(* IEC 61131-3 sources: volt/packages/volt-lsp-iec/test-corpus/lenze-mid/Device/Plc Logic/Application/Library Manager/IODrvEtherCAT, 86 files *)

(* ---- CAA_FILENAME.dut ---- *)
TYPE CAA_FILENAME : CAA.FILENAME;
END_TYPE

(* ---- CAA_PVOID.dut ---- *)
TYPE CAA_PVOID : CAA.PVOID;
END_TYPE

(* ---- CAA_SIZE.dut ---- *)
TYPE CAA_SIZE : CAA.SIZE;
END_TYPE

(* ---- L_ETC_CLEARCOUNTER_COUNTER.dut ---- *)
TYPE L_ETC_CLEARCOUNTER_COUNTER :
(
	NONE := 0,
	COUNTER_MASTER := 1,
	COUNTER_SLAVE := 2,
	COUNTER_ALL := 3
);
END_TYPE

(* ---- L_ETC_CMD_T.dut ---- *)
TYPE L_ETC_CMD_T :
STRUCT
	CMD : UDINT;
	RESULT : UDINT;
END_STRUCT
END_TYPE

(* ---- L_ETC_COE_EMERGENCY.dut ---- *)
TYPE L_ETC_COE_EMERGENCY :
STRUCT
	UIDEVICE : UINT;
	DTTIMESTAMP : DATE_AND_TIME;
	WERRORCODE : WORD;
	BYERRORREGISTER : BYTE;
	ABYDATA : ARRAY [0..4] OF BYTE;
END_STRUCT
END_TYPE

(* ---- L_ETC_COE_EMERGENCY_BUFFER_DATA.dut ---- *)
TYPE L_ETC_COE_EMERGENCY_BUFFER_DATA :
STRUCT
	STRUCTEMERGENCY : L_ETC_COE_EMERGENCY;
	BBUFFEROVERFLOW : BOOL;
END_STRUCT
END_TYPE

(* ---- L_ETC_COE_FLAGS.dut ---- *)
TYPE L_ETC_COE_FLAGS :
(
	ETC_E_COMPLETEACCESS := 16#1
);
END_TYPE

(* ---- L_ETC_DIAGNOSTIC.dut ---- *)
TYPE L_ETC_DIAGNOSTIC :
STRUCT
	WSTATE : L_ETC_STATE;
	STSTATE : STRING;
	XETHERNETLINKUP : BOOL;
	XNOTALLSLAVESOPERATIONAL : BOOL;
	UDIFRAMECOUNTER : UDINT;
	UDIFRAMERESPONSEERRORCOUNTER : UDINT;
	UDICYCWORKINGCOUNTERERRORCOUNTER : UDINT;
	XBUSMISMATCH : BOOL;
	UINUMBEROFSLAVESFOUND : UINT;
	UINUMBEROFSLAVESCONFIGURED : UINT;
	DWLASTERRORCODE : DWORD;
	STLASTERROR : STRING;
	XDC_ENABLED : BOOL;
	XDC_INSYNC : BOOL;
	XDC_BUSY : BOOL;
	DIDC_CURRENTDEVIATION : DINT;
	UDIEMERGENCYNO : UDINT;
END_STRUCT
END_TYPE

(* ---- L_ETC_ENGMODE_STATE.dut ---- *)
TYPE L_ETC_ENGMODE_STATE :
(
	NORMAL := 0,
	ENTERENGMODE := 1,
	ENGMODE := 2,
	LEAVINGENGMODE := 3
);
END_TYPE

(* ---- L_ETC_ERRORCODE.dut ---- *)
TYPE L_ETC_ERRORCODE :
(
	ETC_E_NOERROR := 16#0,
	ETC_E_ERROR := 16#98110000,
	ETC_EMRAS_E_ERROR := 16#98110180,
	ETC_DCM_E_ERROR := 16#981201C0,
	ETC_TEXTBASE := 16#200,
	ETC_ALSTATEBASE := 16#300,
	ETC_E_NOTSUPPORTED := 16#98110001,
	ETC_E_INVALIDINDEX := 16#98110002,
	ETC_E_INVALIDOFFSET := 16#98110003,
	ETC_E_INVALIDSIZE := 16#98110005,
	ETC_E_INVALIDDATA := 16#98110006,
	ETC_E_NOTREADY := 16#98110007,
	ETC_E_BUSY := 16#98110008,
	ETC_E_ACYC_FRM_FREEQ_EMPTY := 16#98110009,
	ETC_E_NOMEMORY := 16#9811000A,
	ETC_E_INVALIDPARM := 16#9811000B,
	ETC_E_NOTFOUND := 16#9811000C,
	ETC_E_INVALIDSTATE := 16#9811000E,
	ETC_E_TIMER_LIST_FULL := 16#9811000F,
	ETC_E_TIMEOUT := 16#98110010,
	ETC_E_OPENFAILED := 16#98110011,
	ETC_E_SENDFAILED := 16#98110012,
	ETC_E_INSERTMAILBOX := 16#98110013,
	ETC_E_INVALIDCMD := 16#98110014,
	ETC_E_UNKNOWN_MBX_PROTOCOL := 16#98110015,
	ETC_E_ACCESSDENIED := 16#98110016,
	ETC_E_PRODKEY_INVALID := 16#9811001A,
	ETC_E_WRONG_FORMAT := 16#9811001B,
	ETC_E_FEATURE_DISABLED := 16#9811001C,
	ETC_E_SHADOW_MEMORY := 16#9811001D,
	ETC_E_BUSCONFIG_MISMATCH := 16#9811001E,
	ETC_E_CONFIGDATAREAD := 16#9811001F,
	ETC_E_XML_CYCCMDS_MISSING := 16#98110021,
	ETC_E_XML_ALSTATUS_READ_MISSING := 16#98110022,
	ETC_E_MCSM_FATAL_ERROR := 16#98110023,
	ETC_E_SLAVE_ERROR := 16#98110024,
	ETC_E_FRAME_LOST := 16#98110025,
	ETC_E_CMD_MISSING := 16#98110026,
	ETC_E_INVALID_DCL_MODE := 16#98110028,
	ETC_E_AI_ADDRESS := 16#98110029,
	ETC_E_INVALID_SLAVE_STATE := 16#9811002A,
	ETC_E_SLAVE_NOT_ADDRESSABLE := 16#9811002B,
	ETC_E_CYC_CMDS_OVERFLOW := 16#9811002C,
	ETC_E_LINK_DISCONNECTED := 16#9811002D,
	ETC_E_MASTERCORE_INACCESSIBLE := 16#9811002E,
	ETC_E_COE_MBXSND_WKC_ERROR := 16#9811002F,
	ETC_E_COE_MBXRCV_WKC_ERROR := 16#98110030,
	ETC_E_NO_MBX_SUPPORT := 16#98110031,
	ETC_E_NO_COE_SUPPORT := 16#98110032,
	ETC_E_NO_EOE_SUPPORT := 16#98110033,
	ETC_E_NO_FOE_SUPPORT := 16#98110034,
	ETC_E_NO_SOE_SUPPORT := 16#98110035,
	ETC_E_NO_VOE_SUPPORT := 16#98110036,
	ETC_E_EVAL_VIOLATION := 16#98110037,
	ETC_E_EVAL_EXPIRED := 16#98110038,
	ETC_E_SDO_ABORTCODE_TOGGLE := 16#98110040,
	ETC_E_SDO_ABORTCODE_TIMEOUT := 16#98110041,
	ETC_E_SDO_ABORTCODE_CCS_SCS := 16#98110042,
	ETC_E_SDO_ABORTCODE_BLK_SIZE := 16#98110043,
	ETC_E_SDO_ABORTCODE_SEQNO := 16#98110044,
	ETC_E_SDO_ABORTCODE_CRC := 16#98110045,
	ETC_E_SDO_ABORTCODE_MEMORY := 16#98110046,
	ETC_E_SDO_ABORTCODE_ACCESS := 16#98110047,
	ETC_E_SDO_ABORTCODE_WRITEONLY := 16#98110048,
	ETC_E_SDO_ABORTCODE_READONLY := 16#98110049,
	ETC_E_SDO_ABORTCODE_INDEX := 16#9811004A,
	ETC_E_SDO_ABORTCODE_PDO_MAP := 16#9811004B,
	ETC_E_SDO_ABORTCODE_PDO_LEN := 16#9811004C,
	ETC_E_SDO_ABORTCODE_P_INCOMP := 16#9811004D,
	ETC_E_SDO_ABORTCODE_I_INCOMP := 16#9811004E,
	ETC_E_SDO_ABORTCODE_HARDWARE := 16#9811004F,
	ETC_E_SDO_ABORTCODE_DATA_SIZE := 16#98110050,
	ETC_E_SDO_ABORTCODE_DATA_SIZE1 := 16#98110051,
	ETC_E_SDO_ABORTCODE_DATA_SIZE2 := 16#98110052,
	ETC_E_SDO_ABORTCODE_OFFSET := 16#98110053,
	ETC_E_SDO_ABORTCODE_DATA_RANGE := 16#98110054,
	ETC_E_SDO_ABORTCODE_DATA_RANGE1 := 16#98110055,
	ETC_E_SDO_ABORTCODE_DATA_RANGE2 := 16#98110056,
	ETC_E_SDO_ABORTCODE_MINMAX := 16#98110057,
	ETC_E_SDO_ABORTCODE_GENERAL := 16#98110058,
	ETC_E_SDO_ABORTCODE_TRANSFER := 16#98110059,
	ETC_E_SDO_ABORTCODE_TRANSFER1 := 16#9811005A,
	ETC_E_SDO_ABORTCODE_TRANSFER2 := 16#9811005B,
	ETC_E_SDO_ABORTCODE_DICTIONARY := 16#9811005C,
	ETC_E_SDO_ABORTCODE_UNKNOWN := 16#9811005D,
	ETC_E_FOE_ERRCODE_NOTDEFINED := 16#98110060,
	ETC_E_FOE_ERRCODE_NOTFOUND := 16#98110061,
	ETC_E_FOE_ERRCODE_ACCESS := 16#98110062,
	ETC_E_FOE_ERRCODE_DISKFULL := 16#98110063,
	ETC_E_FOE_ERRCODE_ILLEGAL := 16#98110064,
	ETC_E_FOE_ERRCODE_PACKENO := 16#98110065,
	ETC_E_FOE_ERRCODE_EXISTS := 16#98110066,
	ETC_E_FOE_ERRCODE_NOUSER := 16#98110067,
	ETC_E_FOE_ERRCODE_BOOTSTRAPONLY := 16#98110068,
	ETC_E_FOE_ERRCODE_NOTINBOOTSTRAP := 16#98110069,
	ETC_E_FOE_ERRCODE_INVALIDPASSWORD := 16#9811006A,
	ETC_E_FOE_ERRCODE_PROGERROR := 16#9811006B,
	ETC_E_CFGFILENOTFOUND := 16#98110070,
	ETC_E_EEPROMREADERROR := 16#98110071,
	ETC_E_EEPROMWRITEERROR := 16#98110072,
	ETC_E_XML_CYCCMDS_SIZEMISMATCH := 16#98110073,
	ETC_E_XML_INVALID_INP_OFF := 16#98110074,
	ETC_E_XML_INVALID_OUT_OFF := 16#98110075,
	ETC_E_PORTCLOSE := 16#98110076,
	ETC_E_PORTOPEN := 16#98110077,
	ETC_E_SOE_ERRORCODE_INVALID_ACCESS := 16#98110078,
	ETC_E_SOE_ERRORCODE_NOT_EXIST := 16#98110079,
	ETC_E_SOE_ERRORCODE_INVL_ACC_ELEM1 := 16#9811007A,
	ETC_E_SOE_ERRORCODE_NAME_NOT_EXIST := 16#9811007B,
	ETC_E_SOE_ERRORCODE_NAME_UNDERSIZE := 16#9811007C,
	ETC_E_SOE_ERRORCODE_NAME_OVERSIZE := 16#9811007D,
	ETC_E_SOE_ERRORCODE_NAME_UNCHANGE := 16#9811007E,
	ETC_E_SOE_ERRORCODE_NAME_WR_PROT := 16#9811007F,
	ETC_E_SOE_ERRORCODE_UNDERS_TRANS := 16#98110080,
	ETC_E_SOE_ERRORCODE_OVERS_TRANS := 16#98110081,
	ETC_E_SOE_ERRORCODE_ATTR_UNCHANGE := 16#98110082,
	ETC_E_SOE_ERRORCODE_ATTR_WR_PROT := 16#98110083,
	ETC_E_SOE_ERRORCODE_UNIT_NOT_EXIST := 16#98110084,
	ETC_E_SOE_ERRORCODE_UNIT_UNDERSIZE := 16#98110085,
	ETC_E_SOE_ERRORCODE_UNIT_OVERSIZE := 16#98110086,
	ETC_E_SOE_ERRORCODE_UNIT_UNCHANGE := 16#98110087,
	ETC_E_SOE_ERRORCODE_UNIT_WR_PROT := 16#98110088,
	ETC_E_SOE_ERRORCODE_MIN_NOT_EXIST := 16#98110089,
	ETC_E_SOE_ERRORCODE_MIN_UNDERSIZE := 16#9811008A,
	ETC_E_SOE_ERRORCODE_MIN_OVERSIZE := 16#9811008B,
	ETC_E_SOE_ERRORCODE_MIN_UNCHANGE := 16#9811008C,
	ETC_E_SOE_ERRORCODE_MIN_WR_PROT := 16#9811008D,
	ETC_E_SOE_ERRORCODE_MAX_NOT_EXIST := 16#9811008E,
	ETC_E_SOE_ERRORCODE_MAX_UNDERSIZE := 16#9811008F,
	ETC_E_SOE_ERRORCODE_MAX_OVERSIZE := 16#98110090,
	ETC_E_SOE_ERRORCODE_MAX_UNCHANGE := 16#98110091,
	ETC_E_SOE_ERRORCODE_MAX_WR_PROT := 16#98110092,
	ETC_E_SOE_ERRORCODE_DATA_NOT_EXIST := 16#98110093,
	ETC_E_SOE_ERRORCODE_DATA_UNDERSIZE := 16#98110094,
	ETC_E_SOE_ERRORCODE_DATA_OVERSIZE := 16#98110095,
	ETC_E_SOE_ERRORCODE_DATA_UNCHANGE := 16#98110096,
	ETC_E_SOE_ERRORCODE_DATA_WR_PROT := 16#98110097,
	ETC_E_SOE_ERRORCODE_DATA_MIN_LIMIT := 16#98110098,
	ETC_E_SOE_ERRORCODE_DATA_MAX_LIMIT := 16#98110099,
	ETC_E_SOE_ERRORCODE_DATA_INCOR := 16#9811009A,
	ETC_E_SOE_ERRORCODE_PASWD_PROT := 16#9811009B,
	ETC_E_SOE_ERRORCODE_TEMP_UNCHANGE := 16#9811009C,
	ETC_E_SOE_ERRORCODE_INVL_INDIRECT := 16#9811009D,
	ETC_E_SOE_ERRORCODE_TEMP_UNCHANGE1 := 16#9811009E,
	ETC_E_SOE_ERRORCODE_ALREADY_ACTIVE := 16#9811009F,
	ETC_E_SOE_ERRORCODE_NOT_INTERRUPT := 16#98110100,
	ETC_E_SOE_ERRORCODE_CMD_NOT_AVAIL := 16#98110101,
	ETC_E_SOE_ERRORCODE_CMD_NOT_AVAIL1 := 16#98110102,
	ETC_E_SOE_ERRORCODE_DRIVE_NO := 16#98110103,
	ETC_E_SOE_ERRORCODE_IDN := 16#98110104,
	ETC_E_SOE_ERRORCODE_FRAGMENT_LOST := 16#98110105,
	ETC_E_SOE_ERRORCODE_BUFFER_FULL := 16#98110106,
	ETC_E_SOE_ERRORCODE_NO_DATA := 16#98110107,
	ETC_E_SOE_ERRORCODE_NO_DEFAULT_VALUE := 16#98110108,
	ETC_E_SOE_ERRORCODE_DEFAULT_LONG := 16#98110109,
	ETC_E_SOE_ERRORCODE_DEFAULT_WP := 16#9811010A,
	ETC_E_SOE_ERRORCODE_INVL_DRIVE_NO := 16#9811010B,
	ETC_E_SOE_ERRORCODE_GENERAL_ERROR := 16#9811010C,
	ETC_E_SOE_ERRCODE_NO_ELEM_ADR := 16#9811010D,
	ETC_E_SLAVE_NOT_PRESENT := 16#9811010E,
	ETC_E_NO_FOE_SUPPORT_BS := 16#9811010F,
	ETC_E_EEPROMRELOADERROR := 16#98110110,
	ETC_E_SLAVECTRLRESETERROR := 16#98110111,
	ETC_E_SYSDRIVERMISSING := 16#98110112,
	ETC_E_BUSCONFIG_TOPOCHANGE := 16#9811011E,
	ETC_E_EOE_MBX_WKC_ERROR := 16#9811011F,
	ETC_E_FOE_MBX_WKC_ERROR := 16#98110120,
	ETC_E_SOE_MBX_WKC_ERROR := 16#98110121,
	ETC_E_AOE_MBX_WKC_ERROR := 16#98110122,
	ETC_E_VOE_MBX_WKC_ERROR := 16#98110123,
	ETC_E_EEPROMASSIGNERROR := 16#98110124,
	ETC_E_MBX_ERROR_TYPE := 16#98110125,
	ETC_DCM_E_NOTINITIALIZED := 16#981201C1,
	ETC_DCM_E_MAX_CTL_ERROR_EXCEED := 16#981201C2,
	ETC_DCM_E_NOMEMORY := 16#981201C3,
	ETC_DCM_E_INVALID_HWLAYER := 16#981201C4,
	ETC_DCM_E_TIMER_MODIFY_ERROR := 16#981201C5,
	ETC_DCM_E_TIMER_NOT_RUNNING := 16#981201C6,
	ETC_DCM_E_WRONG_CPU := 16#981201C7,
	ETC_DCM_E_INVALID_SYNC_PERIOD := 16#981201C8,
	ETC_DCM_E_INVALID_SETVAL := 16#981201C9,
	ETC_DCM_E_DRIFT_TO_HIGH := 16#981201CA,
	ETC_EMRAS_E_INVALIDCOOKIE := 16#98110181,
	ETC_EMRAS_E_MULSRVDISMULCON := 16#98110183,
	ETC_EMRAS_E_LOGONCANCELLED := 16#98110184,
	ETC_EMRAS_E_INVALIDVERSION := 16#98110186,
	ETC_EMRAS_E_INVALIDACCESSCONFIG := 16#98110187,
	ETC_EMRAS_E_ACCESSLESS := 16#98110188,
	ETC_EMRAS_EVT_SERVERSTOPPED := 16#98110191,
	ETC_EMRAS_EVT_WDEXPIRED := 16#98110192,
	ETC_EMRAS_EVT_RECONEXPIRED := 16#98110193,
	ETC_EMRAS_EVT_CLIENTLOGON := 16#98110194,
	ETC_EMRAS_EVT_RECONNECT := 16#98110195,
	ETC_EMRAS_EVT_SOCKCHANGE := 16#98110196,
	ETC_EMRAS_EVT_CLNTDISC := 16#98110197
);
END_TYPE

(* ---- L_ETC_EVTPARAM_PARAMETERTRANSFER.dut ---- *)
TYPE L_ETC_EVTPARAM_PARAMETERTRANSFER :
STRUCT
	WSERVICE : WORD;
	UIDEVICE : WORD;
	DWRESULT : DWORD;
END_STRUCT
END_TYPE

(* ---- L_ETC_HC_GROUPSTATESUMMARY.dut ---- *)
TYPE L_ETC_HC_GROUPSTATESUMMARY :
(
	ETC_STATE_NONE := 16#0,
	ETC_STATE_INIT := 16#1,
	ETC_STATE_PREOPERATIONAL := 16#2,
	ETC_STATE_SAVEOPERATIONAL := 16#4,
	ETC_STATE_OPERATIONAL := 16#8,
	ETC_STATE_SLAVE_MISSING := 16#100,
	ETC_STATE_BOOTSTRAP := 16#700
);
END_TYPE

(* ---- L_ETC_HC_ROLE.dut ---- *)
TYPE L_ETC_HC_ROLE :
(
	HC_ROLE_STATIC := 16#0,
	HC_ROLE_HEAD := 16#1,
	HC_ROLE_MEMBER := 16#2
);
END_TYPE

(* ---- L_ETC_IOCTLOPARMS.dut ---- *)
TYPE L_ETC_IOCTLOPARMS :
STRUCT
	PBYINBUF : POINTER TO BYTE;
	DWINBUFSIZE : DWORD;
	PBYOUTBUF : POINTER TO BYTE;
	DWOUTBUFSIZE : DWORD;
	PDWNUMOUTDATA : POINTER TO DWORD;
END_STRUCT
END_TYPE

(* ---- L_ETC_LANGUAGE.dut ---- *)
TYPE L_ETC_LANGUAGE :
(
	ENG,
	DE
);
END_TYPE

(* ---- L_ETC_MMCSERVICE.dut ---- *)
TYPE L_ETC_MMCSERVICE :
(
	NONE := 0,
	RUN_WITHOUT_CHECK := 16#1,
	RUN_OPTIONAL_SLAVES_ALLOWED := 16#2,
	RUN_OPTIONAL_SLAVES_PROHIBITED := 16#3,
	ADDR_ASSIGNMENT_EXTERNALLY := 16#100,
	ADDR_ASSIGNMENT_CONFIG_SLAVEORDER := 16#200,
	ADDR_ASSIGNMENT_CONFIG_PARAMETER := 16#300
);
END_TYPE

(* ---- L_ETC_MMCSERVICEERROR.dut ---- *)
TYPE L_ETC_MMCSERVICEERROR :
(
	NO_ERROR := 16#0,
	CONFIG_INVALID := 16#1,
	CONFIG_FILE_ERROR := 16#2,
	IDENT_FILE_ERROR := 16#3,
	SERVICE_INVALID := 16#100,
	SERVICE_INVALID_STATE := 16#101,
	ADDR_INTERNAL_ERROR := 16#10000,
	ADDR_NO_MEMORY := 16#10001,
	ADDR_LESS_CONNECTED := 16#10002,
	ADDR_MORE_CONNECTED := 16#10003,
	ADDR_UNEXPECTED_DEVICE := 16#10004,
	ADDR_ASSIGN_ERROR := 16#10005,
	ADDR_NO_SLAVES_CONNECTED := 16#10006
);
END_TYPE

(* ---- L_ETC_MMCSERVICESTATE.dut ---- *)
TYPE L_ETC_MMCSERVICESTATE :
(
	STOPPED,
	RUNNING,
	NOT_READY := 16#FFFF
);
END_TYPE

(* ---- L_ETC_PARAMETERTRANSFERSERVICE_CODE.dut ---- *)
TYPE L_ETC_PARAMETERTRANSFERSERVICE_CODE :
(
	START := WORD#16#1,
	STATE := WORD#16#2,
	DONE := WORD#16#4,
	ABORT := WORD#16#8000
);
END_TYPE

(* ---- L_ETC_SLAVE_PORTS.dut ---- *)
TYPE L_ETC_SLAVE_PORTS :
STRUCT
	PORT0 : BYTE;
	PORT1 : BYTE;
	PORT2 : BYTE;
	PORT3 : BYTE;
END_STRUCT
END_TYPE

(* ---- L_ETC_SLAVE_PORTS2.dut ---- *)
TYPE L_ETC_SLAVE_PORTS2 :
STRUCT
	PORT0 : WORD;
	PORT1 : WORD;
	PORT2 : WORD;
	PORT3 : WORD;
END_STRUCT
END_TYPE

(* ---- L_ETC_SLVSTATISTICS_DESC2_T.dut ---- *)
TYPE L_ETC_SLVSTATISTICS_DESC2_T :
STRUCT
	ABYINVALIDFRAMECNT : ARRAY [0..3] OF BYTE;
	ABYRXERRORCNT : ARRAY [0..3] OF BYTE;
	ABYFWDRXERRORCNT : ARRAY [0..3] OF BYTE;
	BYPROCESSINGUNITERRORCNT : BYTE;
	BYPDIERRORCNT : BYTE;
	WALSTATUSCODE : WORD;
	ABYLOSTLINKCNT : ARRAY [0..3] OF BYTE;
	QWREADTIME : ULINT;
	QWCHANGETIME : ULINT;
END_STRUCT
END_TYPE

(* ---- L_ETC_SLVSTATISTICS_DESC_T.dut ---- *)
TYPE L_ETC_SLVSTATISTICS_DESC_T :
STRUCT
	ABYINVALIDFRAMECNT : ARRAY [0..3] OF BYTE;
	ABYRXERRORCNT : ARRAY [0..3] OF BYTE;
	ABYFWDRXERRORCNT : ARRAY [0..3] OF BYTE;
	BYPROCESSINGUNITERRORCNT : BYTE;
	BYPDIERRORCNT : BYTE;
	WALSTATUSCODE : WORD;
	ABYLOSTLINKCNT : ARRAY [0..3] OF BYTE;
END_STRUCT
END_TYPE

(* ---- L_ETC_STATE.dut ---- *)
TYPE L_ETC_STATE :
(
	ETC_STATE_NONE := 16#0,
	ETC_STATE_INIT := 16#1,
	ETC_STATE_PREOPERATIONAL := 16#2,
	ETC_STATE_BOOT := 16#3,
	ETC_STATE_SAVEOPERATIONAL := 16#4,
	ETC_STATE_OPERATIONAL := 16#8,
	ETC_STATE_UNKNOWN := 16#FFEF
);
END_TYPE

(* ---- ETC_CONSTANTS.gvl ---- *)
VAR_GLOBAL
	_ETC_NUMBER_OF_MASTERS : INT := 1;
	_ETC_NUMBER_OF_SLAVES : INT := 9;
	_ETC_NUMBER_OF_SDO : INT := 676;
	_ETC_NUMBER_OF_INPUT_BYTES : INT := 511;
	_ETC_NUMBER_OF_OUTPUT_BYTES : INT := 511;
	_ETC_SYSTEM_HAS_INTEL_BYTEORDER : BOOL := TRUE;
END_VAR

(* ---- L_ETC_GLOBALS.gvl ---- *)
VAR_GLOBAL
	L_ETC_CMPID_IODRVETC : UDINT := 16#2006;
	L_ETC_EVT_PARAMETERTRANSFER_SERVICE : UDINT := 16#10000003;
END_VAR

(* ---- L_ETC_HC_GROUP_ITF.itf ---- *)
INTERFACE L_ETC_HC_GROUP_ITF
END_INTERFACE

(* ---- GETBOOLEANPROPERTY.pou ---- *)
FUNCTION GETBOOLEANPROPERTY : BOOL
VAR_INPUT
	STKEY : WSTRING;
END_VAR
END_FUNCTION

(* ---- GETCOMPANY.pou ---- *)
FUNCTION GETCOMPANY : WSTRING
END_FUNCTION

(* ---- GETNUMBERPROPERTY.pou ---- *)
FUNCTION GETNUMBERPROPERTY : DINT
VAR_INPUT
	STKEY : WSTRING;
END_VAR
END_FUNCTION

(* ---- GETTEXTPROPERTY.pou ---- *)
FUNCTION GETTEXTPROPERTY : WSTRING
VAR_INPUT
	STKEY : WSTRING;
END_VAR
END_FUNCTION

(* ---- GETTEXTPROPERTY2.pou ---- *)
FUNCTION GETTEXTPROPERTY2 : POINTER TO WSTRING
VAR_INPUT
	STKEY : WSTRING;
END_VAR
END_FUNCTION

(* ---- GETTITLE.pou ---- *)
FUNCTION GETTITLE : WSTRING
END_FUNCTION

(* ---- GETVERSION.pou ---- *)
FUNCTION GETVERSION : VERSION
END_FUNCTION

(* ---- GETVERSIONPROPERTY.pou ---- *)
FUNCTION GETVERSIONPROPERTY : VERSION
VAR_INPUT
	STKEY : WSTRING;
END_VAR
END_FUNCTION

(* ---- L_ETC_GETERRORSTRING.pou ---- *)
FUNCTION L_ETC_GETERRORSTRING : STRING(256)
VAR_INPUT
	EERRORCODE : L_ETC_ERRORCODE;
	ELANGUAGE : L_ETC_LANGUAGE := eng;
END_VAR
END_FUNCTION

(* ---- L_ETC_GETMASTER.pou ---- *)
FUNCTION L_ETC_GETMASTER : POINTER TO L_IODrvEtherCAT
VAR_INPUT
	USICOM : USINT;
END_VAR
END_FUNCTION

(* ---- L_ETC_GETSLAVE.pou ---- *)
FUNCTION L_ETC_GETSLAVE : POINTER TO ETCSlave
VAR_INPUT
	UIDEVICE : UINT;
END_VAR
END_FUNCTION

(* ---- L_ETC_HC_GETGROUP.pou ---- *)
FUNCTION L_ETC_HC_GETGROUP : L_ETC_HC_GROUP_ITF
VAR_INPUT
	USICOM : USINT := 1;
	GROUPNUMBER : UINT;
END_VAR
END_FUNCTION

(* ---- L_ETC_HC_GETGROUPCOUNT.pou ---- *)
FUNCTION L_ETC_HC_GETGROUPCOUNT : UINT
VAR_INPUT
	USICOM : USINT := 1;
END_VAR
END_FUNCTION

(* ---- L_ETC_HC_GETSLAVESOFGROUP.pou ---- *)
FUNCTION L_ETC_HC_GETSLAVESOFGROUP : DWORD
VAR_INPUT
	USICOM : USINT := 1;
	GROUPNUMBER : UINT;
	COUNT : POINTER TO UINT;
	SLAVES : POINTER TO POINTER TO ETCSlave;
END_VAR
END_FUNCTION

(* ---- L_ETC_IOCONTROL.pou ---- *)
FUNCTION L_ETC_IOCONTROL : DWORD
VAR_INPUT
	DWCODE : DWORD;
	PPARMS : POINTER TO L_ETC_IOCTLOPARMS;
END_VAR
END_FUNCTION

(* ---- ETCSLAVE.pou ---- *)
FUNCTION_BLOCK ETCSLAVE
VAR_INPUT
	XSETOPERATIONAL : BOOL;
END_VAR
VAR_OUTPUT
	XDONE : BOOL;
	XBUSY : BOOL;
	XERROR : BOOL;
	EERRORCODE : L_ETC_ERRORCODE;
	WSTATE : WORD;
END_VAR
VAR
	M_PIOCONFIGCONNECTOR : POINTER TO IoConfigConnector;
	M_SZPATH : STRING;
	M_SZNAME : STRING;
	M_DWVENDORID : DWORD;
	M_DWPRODUCTID : DWORD;
	M_DWREVISIONID : DWORD;
	M_UIPHYSSLAVEADDR : UINT;
	M_XDCENABLE : BOOL;
	M_XSETOPERATIONALLAST : BOOL;
	M_WSLAVESTATEACT : WORD;
	FBSLAVE2 : ETCSlave2;
	M_HCINIT : BOOL;
	M_HCINTERFACE : L_ETC_HC_GROUP_ITF;
	M_HCROLE : L_ETC_HC_ROLE;
	M_PMSSELECTIONPAR : POINTER TO IoStandard.IoConfigParameter;
	M_PMSSELECTION : USINT;
	MODULEHANDLERBASE : L_IMHP_ModuleHandler;
	M_SCOMMPATH : STRING(199);
	SLAVEADDRESS : UINT;
	REGISTERONCOMPONENTDIRECTORY : L_IC1P_RegisterOnComponentDirectory;
	M_ITFEVENTCALLBACK : CmpEventMgr.ICmpEventCallback;
	M_HEVENTUPDATECONFIGURATIONDONE : RTS_IEC_HANDLE;
	M_HINTERFACEUPDATECONFIGURATIONDONE : RTS_IEC_HANDLE;
	DCENABLE : BOOL;
	HCGROUP : L_ETC_HC_GROUP_ITF;
	HCROLE : L_ETC_HC_ROLE;
	IODRVETHERCAT : POINTER TO L_IODrvEtherCAT;
	ISMANDATORY : BOOL;
	ISPRESENT : BOOL;
	MODULEHANDLER : L_IMHP_IModuleHandler;
	NAME : STRING;
	PARAMETERSET : USINT;
	PHYSSLAVEADDR : UINT;
	WCSTATE : BOOL;
END_VAR
END_FUNCTION_BLOCK

METHOD EVENTCALLBACK : UDINT
VAR_INPUT
	PEVENTPARAM : POINTER TO EventParam;
END_VAR
END_METHOD

METHOD FB_EXIT : BOOL
VAR_INPUT
	BINCOPYCODE : BOOL;
END_VAR
END_METHOD

METHOD INITIALIZE : UDINT
VAR_INPUT
	WMODULETYPE : UINT;
	DWINSTANCE : UDINT;
	PCONNECTOR : POINTER TO IoConfigConnector;
END_VAR
END_METHOD

METHOD FB_INIT : BOOL
VAR_INPUT
	BINITRETAINS : BOOL;
	BINCOPYCODE : BOOL;
END_VAR
END_METHOD

(* ---- ETCSLAVE2.pou ---- *)
FUNCTION_BLOCK ETCSLAVE2
VAR_INPUT
	XSETOPERATIONAL : BOOL;
END_VAR
VAR_OUTPUT
	XDONE : BOOL;
	XBUSY : BOOL;
	XERROR : BOOL;
	EERRORCODE : L_ETC_ERRORCODE;
	WSTATE : WORD;
END_VAR
VAR
	M_PIOCONFIGCONNECTOR : POINTER TO IoConfigConnector;
	M_XSETOPERATIONALLAST : BOOL;
	M_UIPHYSSLAVEADDR : UINT;
	M_ADWJOBDATA : ARRAY [0..31] OF DWORD;
	GETSTATE : WORD;
	HCGROUP : L_ETC_HC_GROUP_ITF;
	HCROLE : L_ETC_HC_ROLE;
	IODRVETHERCAT : POINTER TO L_IODrvEtherCAT;
	ISMANDATORY : BOOL;
	PHYSSLAVEADDR : UINT;
END_VAR
END_FUNCTION_BLOCK

METHOD INITIALIZE : UDINT
VAR_INPUT
	WMODULETYPE : UINT;
	DWINSTANCE : UDINT;
	PCONNECTOR : POINTER TO IoConfigConnector;
END_VAR
END_METHOD

METHOD SETETCSLAVE
VAR_INPUT
	PCONNECTOR : POINTER TO IoConfigConnector;
	PETCSLAVE : POINTER TO ETCSlave;
END_VAR
END_METHOD

(* ---- ETCSLAVE_DIAG.pou ---- *)
FUNCTION_BLOCK ETCSLAVE_DIAG EXTENDS ETCSlave
VAR
	M_TREE : CAADiagTreeBase;
	CHILDNODECOUNT : CAA.COUNT;
	CONNECTOR : POINTER TO IoStandard.IoConfigConnector;
	ENABLE : BOOL;
	FIRSTCHILDNODE : DED.INode;
	INDEX : UDINT;
	ISROOTNODE : BOOL;
	NEXTSIBLINGNODE : DED.INode;
	PARENTNODE : DED.INode;
	SIBLINGNODECOUNT : CAA.COUNT;
END_VAR
END_FUNCTION_BLOCK

METHOD GETCHILD : DED.INode
VAR_INPUT
	UDIINDEX : UDINT;
END_VAR
END_METHOD

METHOD GETDEVICEDIAGNOSISINFO : DED.ERROR
VAR_INPUT
	PDATA : CAA.PVOID;
	SZSIZE : CAA.SIZE;
END_VAR
VAR_OUTPUT
	SZCOUNT : CAA.SIZE;
END_VAR
END_METHOD

METHOD GETDEVICEERRORASYNC : DED.PROC_STATE
VAR_INPUT
	ECMD : DED.PROC_CMD;
END_VAR
VAR_OUTPUT
	EERROR : DED.ERROR;
END_VAR
VAR_IN_OUT
	ERIDEVICEERROR : DED.ERROR_INFO;
END_VAR
END_METHOD

METHOD GETDEVICEINFO : DED.ERROR
VAR_IN_OUT
	DEIINFO : DED.DEVICE_INFO;
END_VAR
END_METHOD

METHOD GETDEVICESTATE : DED.DEVICE_STATE
VAR_OUTPUT
	XDIAGNOSISINFOAVAILABLE : BOOL;
	EERROR : DED.ERROR;
END_VAR
END_METHOD

METHOD GETSPECIFICDEVICEERRORASYNC : DED.PROC_STATE
VAR_INPUT
	ECMD : DED.PROC_CMD;
	PDATA : CAA.PVOID;
	SZSIZE : CAA.SIZE;
END_VAR
VAR_OUTPUT
	SZCOUNT : CAA.SIZE;
	EERROR : DED.ERROR;
END_VAR
END_METHOD

METHOD GETSPECIFICDEVICESTATE : DED.ERROR
VAR_INPUT
	PDATA : CAA.PVOID;
	SZSIZE : CAA.SIZE;
END_VAR
VAR_OUTPUT
	SZCOUNT : CAA.SIZE;
END_VAR
END_METHOD

METHOD INITIALIZE_DIAG : UDINT
VAR_INPUT
	PCONNECTOR : POINTER TO IoStandard.IoConfigConnector;
	NCONNECTORCOUNT : DINT;
	PARENT : POINTER TO DED.INode;
	CHILDREN : POINTER TO DED.INode;
	UDICHILDCOUNT : UDINT;
END_VAR
END_METHOD

METHOD SETCOMMUNICATIONSTATE : DED.ERROR
VAR_INPUT
	EREQUESTEDSTATE : DED.DEVICE_TRANSITION_STATE;
END_VAR
END_METHOD

(* ---- GLOBALTEXTLIST.pou ---- *)
FUNCTION_BLOCK GLOBALTEXTLIST
VAR
	M_TEXTLISTFILE : STRING(255);
	_STNAMESPACE : STRING;
END_VAR
END_FUNCTION_BLOCK

(* ---- L_ETC_CLEARCOUNTER.pou ---- *)
FUNCTION_BLOCK L_ETC_CLEARCOUNTER
VAR_INPUT
	XEXECUTE : BOOL;
	ECOUNTER : L_ETC_CLEARCOUNTER_COUNTER;
END_VAR
VAR_OUTPUT
	XDONE : BOOL;
	XBUSY : BOOL;
	XERROR : BOOL;
	EERRORCODE : L_ETC_ERRORCODE;
END_VAR
VAR
	XEXECUTELAST : BOOL;
	ADWJOBDATA : ARRAY [0..31] OF DWORD;
END_VAR
END_FUNCTION_BLOCK

(* ---- L_ETC_COE_SDOREAD.pou ---- *)
FUNCTION_BLOCK L_ETC_COE_SDOREAD
VAR_INPUT
	XEXECUTE : BOOL;
	XABORT : BOOL := FALSE;
	USICOM : USINT := 1;
	UIDEVICE : UINT;
	WINDEX : WORD;
	BYSUBINDEX : BYTE;
	UDITIMEOUT : UDINT;
	PBUFFER : CAA_PVOID := 0;
	SZSIZE : CAA_SIZE := 0;
END_VAR
VAR_OUTPUT
	XDONE : BOOL;
	XBUSY : BOOL;
	XERROR : BOOL;
	EERRORCODE : L_ETC_ERRORCODE;
	UDISDOABORT : UDINT;
	SZDATAREAD : CAA_SIZE;
END_VAR
VAR
	XEXECUTELAST : BOOL;
	ADWJOBDATA : ARRAY [0..31] OF DWORD;
END_VAR
END_FUNCTION_BLOCK

(* ---- L_ETC_COE_SDOREAD4.pou ---- *)
FUNCTION_BLOCK L_ETC_COE_SDOREAD4
VAR_INPUT
	XEXECUTE : BOOL;
	XABORT : BOOL := FALSE;
	USICOM : USINT := 1;
	UIDEVICE : UINT;
	WINDEX : WORD;
	BYSUBINDEX : BYTE;
	UDITIMEOUT : UDINT;
END_VAR
VAR_OUTPUT
	XDONE : BOOL;
	XBUSY : BOOL;
	XERROR : BOOL;
	EERRORCODE : L_ETC_ERRORCODE;
	UDISDOABORT : UDINT;
	ABYDATA : ARRAY [0..3] OF BYTE;
	SZDATAREAD : CAA_SIZE;
END_VAR
VAR
	SDOREAD : L_ETC_CoE_SdoRead;
END_VAR
END_FUNCTION_BLOCK

(* ---- L_ETC_COE_SDOREADEX.pou ---- *)
FUNCTION_BLOCK L_ETC_COE_SDOREADEX
VAR_INPUT
	XEXECUTE : BOOL;
	XABORT : BOOL := FALSE;
	USICOM : USINT := 1;
	UIDEVICE : UINT;
	DWFLAGS : DWORD;
	WINDEX : WORD;
	BYSUBINDEX : BYTE;
	UDITIMEOUT : UDINT;
	PBUFFER : CAA_PVOID := 0;
	SZSIZE : CAA_SIZE := 0;
END_VAR
VAR_OUTPUT
	XDONE : BOOL;
	XBUSY : BOOL;
	XERROR : BOOL;
	EERRORCODE : L_ETC_ERRORCODE;
	UDISDOABORT : UDINT;
	SZDATAREAD : CAA_SIZE;
END_VAR
VAR
	XEXECUTELAST : BOOL;
	ADWJOBDATA : ARRAY [0..31] OF DWORD;
END_VAR
END_FUNCTION_BLOCK

(* ---- L_ETC_COE_SDOWRITE.pou ---- *)
FUNCTION_BLOCK L_ETC_COE_SDOWRITE
VAR_INPUT
	XEXECUTE : BOOL;
	XABORT : BOOL := FALSE;
	USICOM : USINT := 1;
	UIDEVICE : UINT;
	WINDEX : WORD;
	BYSUBINDEX : BYTE;
	UDITIMEOUT : UDINT;
	PBUFFER : CAA_PVOID;
	SZSIZE : CAA_SIZE;
END_VAR
VAR_OUTPUT
	XDONE : BOOL;
	XBUSY : BOOL;
	XERROR : BOOL;
	EERRORCODE : L_ETC_ERRORCODE;
	UDISDOABORT : UDINT;
END_VAR
VAR
	XEXECUTELAST : BOOL;
	ADWJOBDATA : ARRAY [0..31] OF DWORD;
END_VAR
END_FUNCTION_BLOCK

(* ---- L_ETC_COE_SDOWRITE4.pou ---- *)
FUNCTION_BLOCK L_ETC_COE_SDOWRITE4
VAR_INPUT
	XEXECUTE : BOOL;
	XABORT : BOOL := FALSE;
	USICOM : USINT := 1;
	UIDEVICE : UINT;
	WINDEX : WORD;
	BYSUBINDEX : BYTE;
	UDITIMEOUT : UDINT;
	ABYDATA : ARRAY [0..3] OF BYTE;
	USIDATALENGTH : USINT;
END_VAR
VAR_OUTPUT
	XDONE : BOOL;
	XBUSY : BOOL;
	XERROR : BOOL;
	EERRORCODE : L_ETC_ERRORCODE;
	UDISDOABORT : UDINT;
END_VAR
VAR
	USILEN : USINT;
	SDOWRITE : L_ETC_CoE_SdoWrite;
END_VAR
END_FUNCTION_BLOCK

(* ---- L_ETC_COE_SDOWRITEEX.pou ---- *)
FUNCTION_BLOCK L_ETC_COE_SDOWRITEEX
VAR_INPUT
	XEXECUTE : BOOL;
	XABORT : BOOL := FALSE;
	USICOM : USINT := 1;
	UIDEVICE : UINT;
	DWFLAGS : DWORD;
	WINDEX : WORD;
	BYSUBINDEX : BYTE;
	UDITIMEOUT : UDINT;
	PBUFFER : CAA_PVOID;
	SZSIZE : CAA_SIZE;
END_VAR
VAR_OUTPUT
	XDONE : BOOL;
	XBUSY : BOOL;
	XERROR : BOOL;
	EERRORCODE : L_ETC_ERRORCODE;
	UDISDOABORT : UDINT;
END_VAR
VAR
	XEXECUTELAST : BOOL;
	ADWJOBDATA : ARRAY [0..31] OF DWORD;
END_VAR
END_FUNCTION_BLOCK

(* ---- L_ETC_ENGINEERINGMODE.pou ---- *)
FUNCTION_BLOCK L_ETC_ENGINEERINGMODE
VAR_INPUT
	USICOM : USINT := 1;
	XENABLE : BOOL;
END_VAR
VAR_OUTPUT
	XBUSY : BOOL;
	XACTIVE : BOOL;
	XERROR : BOOL;
	EERRORCODE : L_ETC_ERRORCODE;
	ESTATE : L_ETC_ENGMODE_STATE;
END_VAR
VAR
	USTEP : UINT := 0;
	XENABLEPRE : BOOL;
	CMD : L_ETC_CMD_T;
	RESULT : DWORD;
	SMSTATE : UDINT;
	FBMASTER : POINTER TO L_IODrvEtherCAT;
END_VAR
END_FUNCTION_BLOCK

(* ---- L_ETC_FOE_READ.pou ---- *)
FUNCTION_BLOCK L_ETC_FOE_READ
VAR_INPUT
	XEXECUTE : BOOL;
	XABORT : BOOL := FALSE;
	USICOM : USINT := 1;
	UIDEVICE : UINT;
	SFILENAME : CAA_FILENAME := '';
	SZFILENAMELEN : CAA_SIZE := 0;
	DWPASSWD : DWORD;
	UDITIMEOUT : UDINT;
	PBUFFER : CAA_PVOID := 0;
	SZSIZE : CAA_SIZE := 0;
END_VAR
VAR_OUTPUT
	XDONE : BOOL;
	XBUSY : BOOL;
	XERROR : BOOL;
	EERRORCODE : L_ETC_ERRORCODE;
	SZDATAREAD : CAA_SIZE;
END_VAR
VAR
	XEXECUTELAST : BOOL;
	ADWJOBDATA : ARRAY [0..31] OF DWORD;
END_VAR
END_FUNCTION_BLOCK

(* ---- L_ETC_FOE_WRITE.pou ---- *)
FUNCTION_BLOCK L_ETC_FOE_WRITE
VAR_INPUT
	XEXECUTE : BOOL;
	XABORT : BOOL := FALSE;
	USICOM : USINT := 1;
	UIDEVICE : UINT;
	SFILENAME : CAA_FILENAME := '';
	SZFILENAMELEN : CAA_SIZE := 0;
	DWPASSWD : DWORD;
	UDITIMEOUT : UDINT;
	PBUFFER : CAA_PVOID := 0;
	SZSIZE : CAA_SIZE := 0;
END_VAR
VAR_OUTPUT
	XDONE : BOOL;
	XBUSY : BOOL;
	XERROR : BOOL;
	EERRORCODE : L_ETC_ERRORCODE;
END_VAR
VAR
	XEXECUTELAST : BOOL;
	ADWJOBDATA : ARRAY [0..31] OF DWORD;
END_VAR
END_FUNCTION_BLOCK

(* ---- L_ETC_GETEMERGENCY.pou ---- *)
FUNCTION_BLOCK L_ETC_GETEMERGENCY
VAR_INPUT
	USICOM : USINT := 1;
	XEXECUTE : BOOL;
	XRESET : BOOL;
END_VAR
VAR_OUTPUT
	XDONE : BOOL;
	XBUSY : BOOL;
	XERROR : BOOL;
	EERRORCODE : L_ETC_ERRORCODE;
	OEMCY : L_ETC_COE_EMERGENCY;
	UICOUNT : UINT;
END_VAR
VAR
	M_XEXECUTELAST : BOOL;
	M_XRESETLAST : BOOL;
END_VAR
END_FUNCTION_BLOCK

METHOD DEINITIALIZE : BOOL
END_METHOD

METHOD FB_INIT : BOOL
VAR_INPUT
	BINITRETAINS : BOOL;
	BINCOPYCODE : BOOL;
END_VAR
END_METHOD

METHOD FB_EXIT : BOOL
VAR_INPUT
	BINCOPYCODE : BOOL;
END_VAR
END_METHOD

METHOD INITIALIZE : BOOL
END_METHOD

(* ---- L_ETC_GETMASTERDIAGNOSTIC.pou ---- *)
FUNCTION_BLOCK L_ETC_GETMASTERDIAGNOSTIC
VAR_INPUT
	XRESET : BOOL;
END_VAR
VAR_OUTPUT
	XDONE : BOOL;
	XBUSY : BOOL;
	XERROR : BOOL;
	EERRORCODE : L_ETC_ERRORCODE;
	ODIAGNOSTIC : L_ETC_DIAGNOSTIC;
END_VAR
VAR
	M_UDILASTMESSAGEID : UDINT;
	M_XRESETLAST : BOOL;
END_VAR
END_FUNCTION_BLOCK

(* ---- L_ETC_GETMASTERSTATE.pou ---- *)
FUNCTION_BLOCK L_ETC_GETMASTERSTATE
VAR_INPUT
	XEXECUTE : BOOL;
	UDITIMEOUT : UDINT;
END_VAR
VAR_OUTPUT
	XDONE : BOOL;
	XBUSY : BOOL;
	XERROR : BOOL;
	EERRORCODE : L_ETC_ERRORCODE;
	WSTATE : WORD;
END_VAR
VAR
	XEXECUTELAST : BOOL;
	ADWJOBDATA : ARRAY [0..31] OF DWORD;
END_VAR
END_FUNCTION_BLOCK

(* ---- L_ETC_GETSLAVESTATE.pou ---- *)
FUNCTION_BLOCK L_ETC_GETSLAVESTATE
VAR_INPUT
	XEXECUTE : BOOL;
	UIDEVICE : UINT;
	UDITIMEOUT : UDINT;
END_VAR
VAR_OUTPUT
	XDONE : BOOL;
	XBUSY : BOOL;
	XERROR : BOOL;
	EERRORCODE : L_ETC_ERRORCODE;
	WSTATE : WORD;
END_VAR
VAR
	XEXECUTELAST : BOOL;
	ADWJOBDATA : ARRAY [0..31] OF DWORD;
END_VAR
END_FUNCTION_BLOCK

METHOD FB_INIT : BOOL
VAR_INPUT
	BINITRETAINS : BOOL;
	BINCOPYCODE : BOOL;
END_VAR
END_METHOD

(* ---- L_ETC_HC_GROUP.pou ---- *)
FUNCTION_BLOCK L_ETC_HC_GROUP
VAR
	M_HDEVMANAGER : RTS_IEC_HANDLE;
	M_HINTERFACE : L_ETC_HC_GROUP_ITF;
	M_USICOM : USINT := 1;
	M_GROUPNUMBER : UINT;
	M_NAME : STRING;
	M_GROUPHEAD : POINTER TO ETCSlave;
	M_IDENTVALUE : UINT;
	M_SLAVECOUNT : UINT;
	M_SLAVES : POINTER TO ETCSlave;
	M_GROUPPRESENT : BOOL;
	M_GROUPSTATESUMMARY : WORD;
	M_WCSTATE : BOOL;
	M_RESERVE : ARRAY [0..15] OF ULINT;
	GETGROUPHEAD : POINTER TO ETCSlave;
	GETGROUPPRESENT : BOOL;
	GETGROUPSTATESUMMARY : L_ETC_HC_GROUPSTATESUMMARY;
	GETIDENTIFICATIONVALUE : UINT;
	GETNAME : STRING;
	GETSLAVECOUNT : UINT;
	GETSLAVES : POINTER TO ETCSlave;
	GROUPHEAD : POINTER TO ETCSlave;
	GROUPNUMBER : UINT;
	GROUPPRESENT : BOOL;
	GROUPSTATESUMMARY : WORD;
	IDENTIFICATIONVALUE : UINT;
	NAME : STRING;
	SLAVECOUNT : UINT;
	SLAVES : POINTER TO ETCSlave;
	WCSTATE : BOOL;
END_VAR
END_FUNCTION_BLOCK

METHOD FB_INIT : BOOL
VAR_INPUT
	BINITRETAINS : BOOL;
	BINCOPYCODE : BOOL;
END_VAR
END_METHOD

METHOD GETGROUPNUMBER : UINT
VAR_INPUT
	HINTERFACE : L_ETC_HC_GROUP_ITF;
END_VAR
END_METHOD

(* ---- L_ETC_HC_SETGROUPSTATE.pou ---- *)
FUNCTION_BLOCK L_ETC_HC_SETGROUPSTATE
VAR_INPUT
	USICOM : USINT := 1;
	XEXECUTE : BOOL;
	UIGROUP : UINT;
	WSTATE : WORD;
	UDITIMEOUT : UDINT;
END_VAR
VAR_OUTPUT
	XDONE : BOOL;
	XBUSY : BOOL;
	XERROR : BOOL;
	EERRORCODE : L_ETC_ERRORCODE;
END_VAR
VAR
	XEXECUTELAST : BOOL;
	ADWJOBDATA : ARRAY [0..31] OF DWORD;
END_VAR
END_FUNCTION_BLOCK

(* ---- L_ETC_HC_SETSLAVEPORTSTATE.pou ---- *)
FUNCTION_BLOCK L_ETC_HC_SETSLAVEPORTSTATE
VAR_INPUT
	USICOM : USINT := 1;
	XEXECUTE : BOOL;
	UIDEVICE : UINT;
	UIPORT : UINT;
	XCLOSE : BOOL;
	XFORCE : BOOL;
	UDITIMEOUT : UDINT;
END_VAR
VAR_OUTPUT
	XDONE : BOOL;
	XBUSY : BOOL;
	XERROR : BOOL;
	EERRORCODE : L_ETC_ERRORCODE;
END_VAR
VAR
	XEXECUTELAST : BOOL;
	ADWJOBDATA : ARRAY [0..16] OF DWORD;
END_VAR
END_FUNCTION_BLOCK

(* ---- L_ETC_MMCASSIGNADDRESS.pou ---- *)
FUNCTION_BLOCK L_ETC_MMCASSIGNADDRESS
VAR_INPUT
	XEXECUTE : BOOL;
	UIPOSITION : UINT;
	UIDEVICE : UINT;
END_VAR
VAR_OUTPUT
	XDONE : BOOL;
	XBUSY : BOOL;
	XERROR : BOOL;
	EERRORCODE : L_ETC_ERRORCODE;
END_VAR
VAR
	FBEEPROMWRITE : L_ETC_WriteEEPROM_intern;
END_VAR
END_FUNCTION_BLOCK

(* ---- L_ETC_MMCCONTROLLER.pou ---- *)
FUNCTION_BLOCK L_ETC_MMCCONTROLLER
VAR_INPUT
	XEXECUTE : BOOL;
	XABORT : BOOL;
	ESERVICE : L_ETC_MMCSERVICE;
	SZCONFIGURATION : STRING;
	XRESETTOPOLOGYCHANGEDCOUNTER : BOOL;
END_VAR
VAR_OUTPUT
	XDONE : BOOL;
	XBUSY : BOOL;
	XERROR : BOOL;
	EERRORCODE : L_ETC_MMCSERVICEERROR;
	XABORTED : BOOL;
	ESERVICESTATE : L_ETC_MMCSERVICESTATE;
	UDITOPOLOGYCHANGEDCOUNTER : UDINT;
END_VAR
VAR
	FBMMC : L_ETC_MMCController_intern;
	ACTUALCONFIGURATION : STRING;
	RUNNINGSERVICE : L_ETC_MMCSERVICE;
END_VAR
END_FUNCTION_BLOCK

METHOD FB_INIT : BOOL
VAR_INPUT
	BINITRETAINS : BOOL;
	BINCOPYCODE : BOOL;
END_VAR
END_METHOD

(* ---- L_ETC_MMCCONTROLLER_INTERN.pou ---- *)
FUNCTION_BLOCK L_ETC_MMCCONTROLLER_INTERN
VAR_INPUT
	XEXECUTE : BOOL;
	XABORT : BOOL;
	ESERVICE : L_ETC_MMCSERVICE;
	SZCONFIGURATION : STRING;
	XRESETTOPOLOGYCHANGEDCOUNTER : BOOL;
END_VAR
VAR_OUTPUT
	XDONE : BOOL;
	XBUSY : BOOL;
	XERROR : BOOL;
	EERRORCODE : L_ETC_MMCSERVICEERROR;
	XABORTED : BOOL;
	ESERVICESTATE : L_ETC_MMCSERVICESTATE;
	UDITOPOLOGYCHANGEDCOUNTER : UDINT;
END_VAR
VAR
	ESERVICEACT : L_ETC_MMCSERVICE;
	SZCONFIGURATIONACT : STRING;
	XEXECUTEPRE : BOOL;
	XABORTPRE : BOOL;
	XRESETTOPOLOGYCHANGEDCOUNTERPRE : BOOL;
	ADATA : ARRAY [0..31] OF DWORD;
END_VAR
END_FUNCTION_BLOCK

METHOD INITIALIZE
END_METHOD

(* ---- L_ETC_MMCCONTROLLERBUS.pou ---- *)
FUNCTION_BLOCK L_ETC_MMCCONTROLLERBUS
VAR_INPUT
	XEXECUTE : BOOL;
	XABORT : BOOL;
	SZCONFIGURATION : STRING;
	ESERVICE : L_ETC_MMCSERVICE;
	XRESETTOPOLOGYCHANGEDCOUNTER : BOOL;
END_VAR
VAR_OUTPUT
	XDONE : BOOL;
	XBUSY : BOOL;
	XERROR : BOOL;
	XABORTED : BOOL;
	EERRORCODE : L_ETC_MMCSERVICEERROR;
	ESERVICESTATE : L_ETC_MMCSERVICESTATE;
	UDITOPOLOGYCHANGEDCOUNTER : UDINT;
END_VAR
VAR
	FBMMC : L_ETC_MMCController;
	POMASTER : POINTER TO L_IODrvEtherCAT;
	STATE : INT;
	XEXECUTELAST : BOOL;
	XABORTLAST : BOOL;
	FBTIMEOUT : TON;
	XREADY : BOOL;
	ACTUALCONFIGURATION : STRING;
	RUNNINGSERVICE : L_ETC_MMCSERVICE;
END_VAR
END_FUNCTION_BLOCK

METHOD RESETOUTPUTS
END_METHOD

METHOD SETOUTPUTS
VAR_INPUT
	EERRORCODE2 : L_ETC_MMCSERVICEERROR;
END_VAR
END_METHOD

(* ---- L_ETC_MMCREADADDRESS.pou ---- *)
FUNCTION_BLOCK L_ETC_MMCREADADDRESS
VAR_INPUT
	XEXECUTE : BOOL;
	UIDEVICE : UINT;
	UDITIMEOUT : UDINT;
END_VAR
VAR_OUTPUT
	XDONE : BOOL;
	XBUSY : BOOL;
	XERROR : BOOL;
	EERRORCODE : L_ETC_ERRORCODE;
	UIDEVICESSA : UINT;
END_VAR
VAR
	FBEEPROMREAD : L_ETC_ReadEEPROM_intern;
END_VAR
END_FUNCTION_BLOCK

(* ---- L_ETC_READEEPROM_INTERN.pou ---- *)
FUNCTION_BLOCK L_ETC_READEEPROM_INTERN
VAR_INPUT
	XEXECUTE : BOOL;
	USICOM : USINT := 1;
	UIDEVICE : UINT;
	BAUTOINCADDR : BOOL := 0;
	UDITIMEOUT : UDINT;
	UIWORDADDRESS : UINT;
	PBUFFER : CAA_PVOID := 0;
	SZSIZE : CAA_SIZE := 0;
END_VAR
VAR_OUTPUT
	XDONE : BOOL;
	XBUSY : BOOL;
	XERROR : BOOL;
	EERRORCODE : L_ETC_ERRORCODE;
	SZDATAREAD : CAA_SIZE;
END_VAR
VAR
	XEXECUTELAST : BOOL;
	ADWJOBDATA : ARRAY [0..31] OF DWORD;
END_VAR
END_FUNCTION_BLOCK

(* ---- L_ETC_READERRCNT.pou ---- *)
FUNCTION_BLOCK L_ETC_READERRCNT
VAR_INPUT
	XEXECUTE : BOOL;
	UIDEVICE : UINT;
END_VAR
VAR_OUTPUT
	XDONE : BOOL;
	XBUSY : BOOL;
	XERROR : BOOL;
	EERRORCODE : L_ETC_ERRORCODE;
	REDERRCNT : L_ETC_SLAVE_PORTS;
	GREENERRCNT : L_ETC_SLAVE_PORTS;
END_VAR
VAR
	WINDEX : WORD;
	XEXCECUTEOLD : BOOL;
	WSTATE : WORD;
	GETSLAVESTATE : L_ETC_GetSlaveState;
	MYEC_T_IOCTLPARMS : L_ETC_IOCTLOPARMS;
	RESULT : DWORD;
	SDOREAD : L_ETC_CoE_SdoRead;
	WMYDATA : WORD;
	DWMYLENGTH : CAA_SIZE := 2;
	BYSUBCODEOFFSET : BYTE;
END_VAR
END_FUNCTION_BLOCK

(* ---- L_ETC_READERRCNT2.pou ---- *)
FUNCTION_BLOCK L_ETC_READERRCNT2
VAR_INPUT
	XEXECUTE : BOOL;
	UIDEVICE : UINT;
END_VAR
VAR_OUTPUT
	XDONE : BOOL;
	XBUSY : BOOL;
	XERROR : BOOL;
	EERRORCODE : L_ETC_ERRORCODE;
	REDERRCNT : L_ETC_SLAVE_PORTS2;
	GREENERRCNT : L_ETC_SLAVE_PORTS;
END_VAR
VAR
	WINDEX : WORD;
	XEXCECUTEOLD : BOOL;
	WSTATE : WORD;
	GETSLAVESTATE : L_ETC_GetSlaveState;
	MYEC_T_IOCTLPARMS : L_ETC_IOCTLOPARMS;
	RESULT : DWORD;
	SDOREAD : L_ETC_CoE_SdoReadEx;
	WMYDATA : WORD;
	DWMYLENGTH : CAA_SIZE := 2;
	BYSUBCODEOFFSET : BYTE;
	EC_SLAVE_BASE_ADDRESS : WORD := 1001;
	EC_IOCTL_FORCE_SLVSTAT_COLLECTION : DWORD := 44;
	EC_SLAVE_CONF_AND_INFO_OBJECT_0X3000 : WORD := 16#3000;
	EC_MOD_BASE_SUBIDX_RX_ERR_CNT_PORT0 : BYTE := 24;
END_VAR
END_FUNCTION_BLOCK

METHOD RESETOUTPUT
END_METHOD

(* ---- L_ETC_READERRCNTREAD.pou ---- *)
FUNCTION_BLOCK L_ETC_READERRCNTREAD
VAR_INPUT
	USICOM : USINT := 1;
	XEXECUTE : BOOL;
	UIDEVICE : UINT;
END_VAR
VAR_OUTPUT
	XDONE : BOOL;
	XBUSY : BOOL;
	XERROR : BOOL;
	EERRORCODE : L_ETC_ERRORCODE;
	RXERRORCNT : L_ETC_SLAVE_PORTS2;
	FWDRXERRORCNT : L_ETC_SLAVE_PORTS;
	PROCESSINGUNITERRORCNT : BYTE;
	PDIERRORCNT : BYTE;
	LOSTLINKCNT : L_ETC_SLAVE_PORTS;
END_VAR
VAR
	XEXCECUTEOLD : BOOL;
	WSTATE : WORD;
	PSLAVE : POINTER TO ETCSlave;
	DWSLAVEID : DWORD;
	SLAVEDESC : L_ETC_SLVSTATISTICS_DESC2_T;
	OIOCTLPARAMS : L_ETC_IOCTLOPARMS;
	RESULT : DWORD;
	DWREAD : DWORD;
	EC_IOCTL_GET_SLVSTATISTICS : DWORD := 45;
END_VAR
END_FUNCTION_BLOCK

METHOD RESETOUTPUT
END_METHOD

(* ---- L_ETC_READERRCNTUPDATE.pou ---- *)
FUNCTION_BLOCK L_ETC_READERRCNTUPDATE
VAR_INPUT
	USICOM : USINT := 1;
	XEXECUTE : BOOL;
END_VAR
VAR_OUTPUT
	XDONE : BOOL;
	XBUSY : BOOL;
	XERROR : BOOL;
	EERRORCODE : L_ETC_ERRORCODE;
END_VAR
VAR
	XEXCECUTEOLD : BOOL;
	WSTATE : WORD;
	PMASTER : POINTER TO L_IODrvEtherCAT;
	UDICYCLETIME : DWORD;
	OIOCTLRPARAMS : L_ETC_IOCTLOPARMS;
	RESULT : DWORD;
	TIMER : TON;
	TVAL : TIME;
	EC_IOCTL_FORCE_SLVSTAT_COLLECTION : DWORD := 44;
END_VAR
END_FUNCTION_BLOCK

METHOD RESETOUTPUTS
END_METHOD

(* ---- L_ETC_REGISTERREAD.pou ---- *)
FUNCTION_BLOCK L_ETC_REGISTERREAD
VAR_INPUT
	XEXECUTE : BOOL;
	XABORT : BOOL := FALSE;
	USICOM : USINT := 1;
	XAUTOINCADDR : BOOL := 0;
	UIDEVICE : UINT;
	WREGISTER : WORD;
	UDITIMEOUT : UDINT;
	PBUFFER : CAA_PVOID := 0;
	SZSIZE : CAA_SIZE := 0;
END_VAR
VAR_OUTPUT
	XDONE : BOOL;
	XBUSY : BOOL;
	XERROR : BOOL;
	EERRORCODE : L_ETC_ERRORCODE;
	SZDATAREAD : CAA_SIZE;
END_VAR
VAR
	XEXECUTELAST : BOOL;
	ADWJOBDATA : ARRAY [0..31] OF DWORD;
END_VAR
END_FUNCTION_BLOCK

(* ---- L_ETC_REGISTERWRITE.pou ---- *)
FUNCTION_BLOCK L_ETC_REGISTERWRITE
VAR_INPUT
	XEXECUTE : BOOL;
	XABORT : BOOL := FALSE;
	USICOM : USINT := 1;
	XAUTOINCADDR : BOOL := 0;
	UIDEVICE : UINT;
	WREGISTER : WORD;
	UDITIMEOUT : UDINT;
	PBUFFER : CAA_PVOID := 0;
	SZSIZE : CAA_SIZE := 0;
END_VAR
VAR_OUTPUT
	XDONE : BOOL;
	XBUSY : BOOL;
	XERROR : BOOL;
	EERRORCODE : L_ETC_ERRORCODE;
END_VAR
VAR
	XEXECUTELAST : BOOL;
	ADWJOBDATA : ARRAY [0..31] OF DWORD;
END_VAR
END_FUNCTION_BLOCK

(* ---- L_ETC_RESETERRCNT.pou ---- *)
FUNCTION_BLOCK L_ETC_RESETERRCNT
VAR_INPUT
	XEXECUTE : BOOL;
END_VAR
VAR_OUTPUT
	XDONE : BOOL;
	XBUSY : BOOL;
	XERROR : BOOL;
	EERRORCODE : L_ETC_ERRORCODE;
END_VAR
VAR
	XEXCECUTEOLD : BOOL := 0;
	WSTATE : WORD;
	GETMASTERSTATE : L_ETC_GetMasterState;
	MYEC_T_IOCTLPARMS : L_ETC_IOCTLOPARMS;
	RESULT : DWORD := 0;
END_VAR
END_FUNCTION_BLOCK

(* ---- L_ETC_SETMASTERSTATE.pou ---- *)
FUNCTION_BLOCK L_ETC_SETMASTERSTATE
VAR_INPUT
	XEXECUTE : BOOL;
	WSTATE : WORD;
	UDITIMEOUT : UDINT;
END_VAR
VAR_OUTPUT
	XDONE : BOOL;
	XBUSY : BOOL;
	XERROR : BOOL;
	EERRORCODE : L_ETC_ERRORCODE;
END_VAR
VAR
	XEXECUTELAST : BOOL;
	ADWJOBDATA : ARRAY [0..31] OF DWORD;
END_VAR
END_FUNCTION_BLOCK

(* ---- L_ETC_SETSLAVESTATE.pou ---- *)
FUNCTION_BLOCK L_ETC_SETSLAVESTATE
VAR_INPUT
	XEXECUTE : BOOL;
	UIDEVICE : UINT;
	WSTATE : WORD;
	UDITIMEOUT : UDINT;
END_VAR
VAR_OUTPUT
	XDONE : BOOL;
	XBUSY : BOOL;
	XERROR : BOOL;
	EERRORCODE : L_ETC_ERRORCODE;
END_VAR
VAR
	XEXECUTELAST : BOOL;
	ADWJOBDATA : ARRAY [0..31] OF DWORD;
END_VAR
END_FUNCTION_BLOCK

(* ---- L_ETC_SETSLAVESTATEFWDL.pou ---- *)
FUNCTION_BLOCK L_ETC_SETSLAVESTATEFWDL
VAR_INPUT
	XEXECUTE : BOOL;
	UIDEVICE : UINT;
	WSTATE : WORD;
	UDITIMEOUT : UDINT;
END_VAR
VAR_OUTPUT
	XDONE : BOOL;
	XBUSY : BOOL;
	XERROR : BOOL;
	EERRORCODE : L_ETC_ERRORCODE;
END_VAR
VAR
	XEXECUTELAST : BOOL;
	ADWJOBDATA : ARRAY [0..31] OF DWORD;
END_VAR
END_FUNCTION_BLOCK

(* ---- L_ETC_VOE_WRITEREAD_INTERN.pou ---- *)
FUNCTION_BLOCK L_ETC_VOE_WRITEREAD_INTERN
VAR_INPUT
	XEXECUTE : BOOL;
	USICOM : USINT := 1;
	UIDEVICE : UINT;
	UDITIMEOUT : UDINT;
	USICHANNEL : USINT;
	UDIVENDORID : UDINT;
	UIVENDORTYPE : UINT;
	PBUFFERWRITE : CAA_PVOID;
	SZSIZEWRITE : CAA_SIZE;
	PBUFFERREAD : CAA_PVOID;
	SZSIZEREAD : CAA_SIZE;
END_VAR
VAR_OUTPUT
	XDONE : BOOL;
	XBUSY : BOOL;
	XERROR : BOOL;
	EERRORCODE : L_ETC_ERRORCODE;
	SZDATAREAD : CAA_SIZE;
END_VAR
VAR
	XEXECUTELAST : BOOL;
	ADWJOBDATA : ARRAY [0..31] OF DWORD;
END_VAR
END_FUNCTION_BLOCK

(* ---- L_ETC_WRITEEEPROM_INTERN.pou ---- *)
FUNCTION_BLOCK L_ETC_WRITEEEPROM_INTERN
VAR_INPUT
	XEXECUTE : BOOL;
	USICOM : USINT := 1;
	UIDEVICE : UINT;
	BAUTOINCADDR : BOOL := 0;
	UDITIMEOUT : UDINT;
	UIWORDADDRESS : UINT;
	PBUFFER : CAA_PVOID := 0;
	SZSIZE : CAA_SIZE := 0;
END_VAR
VAR_OUTPUT
	XDONE : BOOL;
	XBUSY : BOOL;
	XERROR : BOOL;
	EERRORCODE : L_ETC_ERRORCODE;
END_VAR
VAR
	XEXECUTELAST : BOOL;
	ADWJOBDATA : ARRAY [0..31] OF DWORD;
END_VAR
END_FUNCTION_BLOCK

(* ---- L_IODRVETHERCAT.pou ---- *)
FUNCTION_BLOCK L_IODRVETHERCAT
VAR_INPUT
	XRESTART : BOOL := FALSE;
	XSTOPBUS : BOOL := FALSE;
	XWAITWHILEBOOTINGCONTINUE : BOOL;
END_VAR
VAR_OUTPUT
	XDONE : BOOL;
	XBUSY : BOOL;
	XERROR : BOOL;
	EERRORCODE : L_ETC_ERRORCODE;
	WSTATE : WORD;
	XDISTRIBUTEDCLOCKINSYNC : BOOL;
	XWAITWHILEBOOTING : BOOL;
END_VAR
VAR
	M_PIOCONFIGCONNECTOR : POINTER TO IoConfigConnector;
	M_FBIODRVETHERCAT : L_IODrvEtherCAT_intern2;
	M_UDICYCLETIME : UDINT;
	M_NUMBEROFSLAVESCONFIGURED : UINT;
	M_IDX_NEXT : UINT;
	M_IDX_CHUNK : UINT := 3;
	MODULEHANDLERBASE : L_IMHP_ModuleHandler;
	CYCLETIME : UDINT;
	GETCONNECTOR : POINTER TO IoConfigConnector;
	MODULEHANDLER : L_IMHP_IModuleHandler;
	NUMBEROFSLAVESCONFIGURED : UINT;
	WCSTATE : BOOL;
END_VAR
END_FUNCTION_BLOCK

METHOD BEFOREREADINPUTS
END_METHOD

METHOD INITIALIZE : UDINT
VAR_INPUT
	WMODULETYPE : UINT;
	DWINSTANCE : UDINT;
	PCONNECTOR : POINTER TO IoConfigConnector;
END_VAR
END_METHOD

METHOD FB_INIT : BOOL
VAR_INPUT
	BINITRETAINS : BOOL;
	BINCOPYCODE : BOOL;
END_VAR
END_METHOD

(* ---- L_IODRVETHERCAT_DIAG.pou ---- *)
FUNCTION_BLOCK L_IODRVETHERCAT_DIAG EXTENDS L_IODrvEtherCAT
VAR
	M_TREE : CAADiagTreeBase;
	M_DIAG : L_ETC_GetMasterDiagnostic;
	CHILDNODECOUNT : CAA.COUNT;
	CONNECTOR : POINTER TO IoStandard.IoConfigConnector;
	ENABLE : BOOL;
	FIRSTCHILDNODE : DED.INode;
	INDEX : UDINT;
	ISROOTNODE : BOOL;
	NEXTSIBLINGNODE : DED.INode;
	PARENTNODE : DED.INode;
	SIBLINGNODECOUNT : CAA.COUNT;
END_VAR
END_FUNCTION_BLOCK

METHOD GETBUSDIAGNOSISINFO : DED.ERROR
VAR_INPUT
	PDATA : CAA.PVOID;
	SZSIZE : CAA.SIZE;
END_VAR
VAR_OUTPUT
	SZCOUNT : CAA.SIZE;
END_VAR
END_METHOD

METHOD GETBUSERRORASYNC : DED.PROC_STATE
VAR_INPUT
	ECMD : DED.PROC_CMD;
END_VAR
VAR_OUTPUT
	EERROR : DED.ERROR;
END_VAR
VAR_IN_OUT
	ERIBUSERROR : DED.ERROR_INFO;
END_VAR
END_METHOD

METHOD GETBUSINFO : DED.ERROR
VAR_IN_OUT
	BUIINFO : DED.BUS_INFO;
END_VAR
END_METHOD

METHOD GETBUSSTATE : DED.BUS_STATE
VAR_OUTPUT
	XDIAGNOSISINFOAVAILABLE : BOOL;
	EERROR : DED.ERROR;
END_VAR
END_METHOD

METHOD GETCHILD : DED.INode
VAR_INPUT
	UDIINDEX : UDINT;
END_VAR
END_METHOD

METHOD GETDEVICEDIAGNOSISINFO : DED.ERROR
VAR_INPUT
	PDATA : CAA.PVOID;
	SZSIZE : CAA.SIZE;
END_VAR
VAR_OUTPUT
	SZCOUNT : CAA.SIZE;
END_VAR
END_METHOD

METHOD GETDEVICEERRORASYNC : DED.PROC_STATE
VAR_INPUT
	ECMD : DED.PROC_CMD;
END_VAR
VAR_OUTPUT
	EERROR : DED.ERROR;
END_VAR
VAR_IN_OUT
	ERIDEVICEERROR : DED.ERROR_INFO;
END_VAR
END_METHOD

METHOD GETDEVICEINFO : DED.ERROR
VAR_IN_OUT
	DEIINFO : DED.DEVICE_INFO;
END_VAR
END_METHOD

METHOD GETDEVICESTATE : DED.DEVICE_STATE
VAR_OUTPUT
	XDIAGNOSISINFOAVAILABLE : BOOL;
	EERROR : DED.ERROR;
END_VAR
END_METHOD

METHOD GETQOS : DED.ERROR
VAR_IN_OUT
	QUALITYINFO : DED.QOS_INFO;
END_VAR
END_METHOD

METHOD GETSPECIFICBUSSTATE : DED.ERROR
VAR_INPUT
	PDATA : CAA.PVOID;
	SZSIZE : CAA.SIZE;
END_VAR
VAR_OUTPUT
	SZCOUNT : CAA.SIZE;
END_VAR
END_METHOD

METHOD GETSPECIFICDEVICEERRORASYNC : DED.PROC_STATE
VAR_INPUT
	ECMD : DED.PROC_CMD;
	PDATA : CAA.PVOID;
	SZSIZE : CAA.SIZE;
END_VAR
VAR_OUTPUT
	SZCOUNT : CAA.SIZE;
	EERROR : DED.ERROR;
END_VAR
END_METHOD

METHOD GETSPECIFICDEVICESTATE : DED.ERROR
VAR_INPUT
	PDATA : CAA.PVOID;
	SZSIZE : CAA.SIZE;
END_VAR
VAR_OUTPUT
	SZCOUNT : CAA.SIZE;
END_VAR
END_METHOD

METHOD INITIALIZE_DIAG : UDINT
VAR_INPUT
	PCONNECTOR : POINTER TO IoStandard.IoConfigConnector;
	NCONNECTORCOUNT : DINT;
	PARENT : POINTER TO DED.INode;
	CHILDREN : POINTER TO DED.INode;
	UDICHILDCOUNT : UDINT;
END_VAR
END_METHOD

METHOD SETCOMMUNICATIONSTATE : DED.ERROR
VAR_INPUT
	EREQUESTEDSTATE : DED.DEVICE_TRANSITION_STATE;
END_VAR
END_METHOD

(* ---- L_IODRVETHERCAT_INTERN.pou ---- *)
FUNCTION_BLOCK L_IODRVETHERCAT_INTERN
VAR_INPUT
	XRESTART : BOOL := FALSE;
	XSTOPBUS : BOOL := FALSE;
END_VAR
VAR_OUTPUT
	XDONE : BOOL;
	XBUSY : BOOL;
	XERROR : BOOL;
	EERRORCODE : L_ETC_ERRORCODE;
	WSTATE : WORD;
	XDISTRIBUTEDCLOCKINSYNC : BOOL;
END_VAR
VAR
	M_PIOCONFIGCONNECTOR : POINTER TO IoConfigConnector;
	M_WCOMMAND : UDINT;
	M_UDISTOPTIMEOUT : UDINT := 5000;
	M_UDISTARTTIMEOUT : UDINT := 60000;
	M_UDILASTMESSAGEID : UDINT;
	M_SLASTMESSAGE : STRING;
	M_WSTATEREQ : UINT;
	M_ADWJOBDATA : ARRAY [0..31] OF DWORD;
	M_XRESTARTLAST : BOOL;
	M_XSTOPBUSLAST : BOOL;
	NUMBEROFSLAVESCONFIGURED : UINT;
	WCSTATE : BOOL;
END_VAR
END_FUNCTION_BLOCK

METHOD BEFOREREADINPUTS
END_METHOD

METHOD INITIALIZE : UDINT
VAR_INPUT
	WMODULETYPE : UINT;
	DWINSTANCE : UDINT;
	PCONNECTOR : POINTER TO IoConfigConnector;
	PPARENT : POINTER TO L_IODrvEtherCAT;
END_VAR
END_METHOD

(* ---- L_IODRVETHERCAT_INTERN2.pou ---- *)
FUNCTION_BLOCK L_IODRVETHERCAT_INTERN2
VAR_INPUT
	XRESTART : BOOL := FALSE;
	XSTOPBUS : BOOL := FALSE;
	XWAITWHILEBOOTINGCONTINUE : BOOL;
	DWRESERVEINPUT : ARRAY [0..15] OF DWORD;
END_VAR
VAR_OUTPUT
	XDONE : BOOL;
	XBUSY : BOOL;
	XERROR : BOOL;
	EERRORCODE : L_ETC_ERRORCODE;
	WSTATE : WORD;
	XDISTRIBUTEDCLOCKINSYNC : BOOL;
	XWAITWHILEBOOTING : BOOL;
	DWRESERVEOUTPUT : ARRAY [0..15] OF DWORD;
END_VAR
VAR
	M_PIOCONFIGCONNECTOR : POINTER TO IoConfigConnector;
	M_WCOMMAND : UDINT;
	M_UDISTOPTIMEOUT : UDINT := 5000;
	M_UDISTARTTIMEOUT : UDINT := 60000;
	M_UDILASTMESSAGEID : UDINT;
	M_SLASTMESSAGE : STRING;
	M_WSTATEREQ : UINT;
	M_ADWJOBDATA : ARRAY [0..31] OF DWORD;
	M_XRESTARTLAST : BOOL;
	M_XSTOPBUSLAST : BOOL;
	DWRESERVEMEM : ARRAY [0..15] OF DWORD;
	NUMBEROFSLAVESCONFIGURED : UINT;
	WCSTATE : BOOL;
END_VAR
END_FUNCTION_BLOCK

METHOD BEFOREREADINPUTS
END_METHOD

METHOD INITIALIZE : UDINT
VAR_INPUT
	WMODULETYPE : UINT;
	DWINSTANCE : UDINT;
	PCONNECTOR : POINTER TO IoConfigConnector;
	PPARENT : POINTER TO L_IODrvEtherCAT;
END_VAR
END_METHOD
